FUNCTION_BLOCK SQRT_REAL (* IEC 61131-3,Table 23#2 *)
  (* Standard: 61131-3 *)
  (* Version 0.1, 2006-09-12, JHC, Holobloc Inc, Converted to Template. *)
  (* Version 0.0, 2004-12-15, JHC, Rockwell Automation, Converted from SRC format. *)
  (* Compiler header: package fb.rt.plc.math; *)
  (* Compiler classdef: (Math.sqrt( IN )) *)
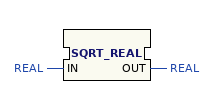
  VAR_INPUT
    IN : REAL;
  END_VAR
  VAR_OUTPUT
    OUT : REAL;
  END_VAR
END_FUNCTION_BLOCK
